{attribute 'GeneratedUsingTerminal: EL1918-0000-0016'}
{attribute addProperty BoxType "EL1918-0000-0016"}
{attribute addProperty Id "FSoE_CommandUSINT1FSIN_Module_1_InputBOOL1FSIN_Module_1_Module_FaultBOOL1FSIN_Module_2_InputBOOL1FSIN_Module_2_Module_FaultBOOL1FSIN_Module_3_InputBOOL1FSIN_Module_3_Module_FaultBOOL1FSIN_Module_4_InputBOOL1FSIN_Module_4_Module_FaultBOOL1FSIN_Module_5_InputBOOL1FSIN_Module_5_Module_FaultBOOL1FSIN_Module_6_InputBOOL1FSIN_Module_6_Module_FaultBOOL1FSIN_Module_7_InputBOOL1FSIN_Module_7_Module_FaultBOOL1FSIN_Module_8_InputBOOL1FSIN_Module_8_Module_FaultBOOL1FSoE_CRC_000UINT2FSoE_Connection_IDUINT2"}
{attribute addProperty CRC "2352904646"}
{attribute addProperty Size "21"}
TYPE FSOE_8C3E79C6 :
STRUCT
	{attribute addProperty Name "FSoE_Command"}
	FSoE_Command : USINT;
	{attribute addProperty Name "FSIN_Module_1_Input"}
	FSIN_Module_1_Input : BOOL;
	{attribute addProperty Name "FSIN_Module_1_Module_Fault"}
	FSIN_Module_1_Module_Fault : BOOL;
	{attribute addProperty Name "FSIN_Module_2_Input"}
	FSIN_Module_2_Input : BOOL;
	{attribute addProperty Name "FSIN_Module_2_Module_Fault"}
	FSIN_Module_2_Module_Fault : BOOL;
	{attribute addProperty Name "FSIN_Module_3_Input"}
	FSIN_Module_3_Input : BOOL;
	{attribute addProperty Name "FSIN_Module_3_Module_Fault"}
	FSIN_Module_3_Module_Fault : BOOL;
	{attribute addProperty Name "FSIN_Module_4_Input"}
	FSIN_Module_4_Input : BOOL;
	{attribute addProperty Name "FSIN_Module_4_Module_Fault"}
	FSIN_Module_4_Module_Fault : BOOL;
	{attribute addProperty Name "FSIN_Module_5_Input"}
	FSIN_Module_5_Input : BOOL;
	{attribute addProperty Name "FSIN_Module_5_Module_Fault"}
	FSIN_Module_5_Module_Fault : BOOL;
	{attribute addProperty Name "FSIN_Module_6_Input"}
	FSIN_Module_6_Input : BOOL;
	{attribute addProperty Name "FSIN_Module_6_Module_Fault"}
	FSIN_Module_6_Module_Fault : BOOL;
	{attribute addProperty Name "FSIN_Module_7_Input"}
	FSIN_Module_7_Input : BOOL;
	{attribute addProperty Name "FSIN_Module_7_Module_Fault"}
	FSIN_Module_7_Module_Fault : BOOL;
	{attribute addProperty Name "FSIN_Module_8_Input"}
	FSIN_Module_8_Input : BOOL;
	{attribute addProperty Name "FSIN_Module_8_Module_Fault"}
	FSIN_Module_8_Module_Fault : BOOL;
	{attribute addProperty Name "FSoE_CRC_000"}
	FSoE_CRC_000 : UINT;
	{attribute addProperty Name "FSoE_Connection_ID"}
	FSoE_Connection_ID : UINT;
END_STRUCT
END_TYPE

(* stored: Version 1.2.0.0, ProductVersion 3.1.4024.9
   DUT FSOE_8C3E79C6: Id {1a9ceef6-d24d-4956-bf00-081624211506} *)
